{attribute 'qualified_only'}
VAR_GLOBAL RETAIN
	configValues				:   ST_ConfigValues;		// Konfigurationsparaeter - Müssen vom User geändert werden können
END_VAR

(* stored: Version 1.1.0.1
   GVL GVL: Id {5aaa212f-5667-440f-b23e-01d8197849cd} *)
